PROGRAM MAIN
VAR
	pbGapMode: BOOL:=FALSE;
	pbTaperMode: BOOL:=FALSE;
	pbSingleCarrierMode: BOOL:=FALSE;
	pbDebugMode:BOOL:=FALSE;
	pbBCGapMode:BOOL:=FALSE;
	fb_led_Show: FB_LedShow;
	btn_reset: BOOL;
	CPMU_PLC_Reset: PLC_Reset;
	d_state: DINT;
	CPMU_PLC_Start: PLC_Start;
	powerStatus:BOOL;

(*TwinSAFE*)
	Safe_run AT%Q*:BOOL;
	Err_Ack AT %Q*:BOOL;
	Estop_RunAndRestart AT %Q*:BOOL;
	AX5805_Error_Ack AT %Q*:BOOL;
	Led_Run  AT %Q*:BOOL;
	Led_Error  AT %Q*:BOOL;

	FB_ERROR AT%I*:BOOL;
	COM_ERROR AT%I*:BOOL;
	//OUT_ERROR AT%I*:BOOL;
	Estop_Out AT%I*:BOOL;

	SafeStatus:INT;
	SafePLCRunOK: BOOL;
	fb_ton: TON;
	fb_ton2: TON;
	fb_ton3: TON;
	fb_ton1: TON;
	fb_ton0: TON;
(*IO*)
	el1808_D1  AT%I* :ARRAY[1..8] OF BOOL;
	el1008 AT%I*:BOOL;
	EStopTrig:BOOL;
(*setAxisPosition*)
	SetAxisPosState: INT;
	FB_Set_AxisPosition:FB_SetAxisPosition;
	fb_ton4: TON;
	fb_ton5: TON;
	fb_ton6: TON;
	SerAxisPositionDone: BOOL;

	i: INT;
	j: INT;

(****RS232***)
	fbEL6001	: FB_SerialCom;
	moveDoneLeftTop: BOOL;
	moveDoneRightTop: BOOL;
	moveDoneLeftBottom: BOOL;
	moveDoneRightBottom: BOOL;
	moveDoneAllAxis: BOOL;
	moveStatusLeftTop: BOOL;
	moveStatusRightTop: BOOL;
	moveStatusLeftBottom: BOOL;
	moveStatusRightBottom: BOOL;
	moveStatusAllAxis: BOOL;

(*Torque*)
	Torque_LT AT%I*:INT;
	Torque_RT AT%I*:INT;
	Torque_LB AT%I*:INT;
	Torque_RB AT%I*:INT;
(**)
	btn_setAxisPosition: BOOL;
	ValueSet_LeftTop:LREAL;
	ValueSet_RightTop:LREAL;
	ValueSet_LeftBottom:LREAL;
	ValueSet_RightBottom:LREAL;
(**)
	RestartTC: TC_Restart;
	
(*recipe*)
	RecipeINT:INT;
	RecipeBOOL:BOOL;
	RecipeManCommands: RecipeManCommands;
	SaveParameter : BOOL;  //保存文件
	LoadParameter : BOOL;  //读取文件
	Save_R_TRIG   : R_TRIG;
	Read_R_TRIG   : R_TRIG;
	loadparameterStatus: INT;
	RecipeBOOL2:BOOL;
	ReturnDwordLoad: DWORD;
	InsertionDeviceName:STRING;
(*UserMode*)
	pbUserMode: BOOL:=TRUE;
	EL1904 AT%I* :ARRAY[1..24] OF BOOL;
	setAxisPositionEnable: BOOL;
	state_loadParameters: INT;
	state_setLEPosBias: INT;
	//
	PositionBiasSet:BOOL;
	MC_SetLEPosBias_LeftTop:MC_WriteParameter;
	MC_SetLEPosBias_RightTop:MC_WriteParameter;
	MC_SetLEPosBias_LeftBottom:MC_WriteParameter;
	MC_SetLEPosBias_RightBottom:MC_WriteParameter;
	PositionBias_LeftTop: LREAL:=10.1;
	PositionBias_RightTop: LREAL:=10.2;
	PositionBias_LeftBottom: LREAL:=10.3;
	PositionBias_RightBottom: LREAL:=10.4;

	LoadLEPB_R_TRIG: R_TRIG;
	PositionBiasTON: TON;
	
	//
	OPC_TEST_Bi:BOOL:=TRUE; (*~ (OPC:1:available for OPC Clients) *)
	OPC_TEST_Bi2:BOOL;(*~ (OPC:1:available for OPC Clients) *)
	//
	HasTemperatureSensorOrNot:BOOL;//Only IVU or CPMU
	(*Sensor Reading*)
	Sensor_Reading_1 AT %I*:ARRAY[0..3] OF BYTE;
	Sensor_Reading_2 AT %I*:ARRAY[0..3] OF BYTE;
	Sensor_Reading_3 AT %I*:ARRAY[0..3] OF BYTE;
	Sensor_Reading_4 AT %I*:ARRAY[0..3] OF BYTE;
	Sensor_Reading_5 AT %I*:ARRAY[0..3] OF BYTE;
	Sensor_Reading_6 AT %I*:ARRAY[0..3] OF BYTE;
	Sensor_Reading_7 AT %I*:ARRAY[0..3] OF BYTE;
	Sensor_Reading_8 AT %I*:ARRAY[0..3] OF BYTE;
	Sensor_Reading_DpState AT %I*:USINT;
	Sensor_Reading_ExtDiagFlag AT %I*:BOOL;
	TemperatureSensors_1:LREAL;
	TemperatureSensors_2:LREAL;
	TemperatureSensors_3:LREAL;
	TemperatureSensors_4:LREAL;
	TemperatureSensors_5:LREAL;
	TemperatureSensors_6:LREAL;
	TemperatureSensors_7:LREAL;
	TemperatureSensors_8:LREAL;
	dut_sensor_datas_1:DUT_SENSOR_DATAS_1;
	dut_sensor_datas_2:DUT_SENSOR_DATAS_2;
	dut_sensor_datas_3:DUT_SENSOR_DATAS_3;
	dut_sensor_datas_4:DUT_SENSOR_DATAS_4;
	dut_sensor_datas_5:DUT_SENSOR_DATAS_5;
	dut_sensor_datas_6:DUT_SENSOR_DATAS_6;
	dut_sensor_datas_7:DUT_SENSOR_DATAS_7;
	dut_sensor_datas_8:DUT_SENSOR_DATAS_8;
	//
	temperature_gradient_2_To_1:LREAL;
	temperature_gradient_3_To_2:LREAL;
	temperature_gradient_5_To_4:LREAL;
	temperature_gradient_6_To_5:LREAL;
	temperature_gradient_max:LREAL;
	//
	temperature_average:LREAL;
	A_SetLinearEncoderPositionBias_Enable: BOOL;
	
		//
	temperatureStatus:INT;//0：有传感器度数错误；1:常温；2:低温；3:常温和低温中间态
	CryogenicTemperatureThreshold:LREAL:=80;//80K以下归划分为低温
	RoomTemperatureThreshold:LREAL:=293;//293K以上划分为常温
	//CPMU cryogenix ON/FF
	CryogenicCompensationOn:BOOL;
	CryogenicCompensationConditionsReady:BOOL;
	CryogenicCompensation_LeftTop:LREAL;
	CryogenicCompensation_RightTop:LREAL;
	CryogenicCompensation_LeftBottom:LREAL;
	CryogenicCompensation_RightBottom:LREAL;
	CryogenicCompensationDone: BOOL;
	
	(**)
	bDriveDiagMessageAndNumber  : BOOL;
	m_GetDriveStatusState:INT;
	GetDriveStatusStateDone:BOOL;
	GetDriveStatusStateError:BOOL;
	GetDriveStatusTON: TON;
	//	
	fb_SoEReadDiagMessage_LeftTop: FB_SoEReadDiagMessage;
	fb_SoEReadDiagMessage_RightTop: FB_SoEReadDiagMessage;
	fb_SoEReadDiagMessage_LeftBottom: FB_SoEReadDiagMessage;
	fb_SoEReadDiagMessage_RightBottom: FB_SoEReadDiagMessage;
	DriveDiagMessage_LeftTop:STRING;
	DriveDiagMessage_RightTop:STRING;
	DriveDiagMessage_LeftBottom:STRING;
	DriveDiagMessage_RightBottom:STRING;
	//
	FB_SoEReadDiagNumber_LeftTop: FB_SoEReadDiagNumber;
	FB_SoEReadDiagNumber_RightTop: FB_SoEReadDiagNumber;
	FB_SoEReadDiagNumber_LeftBottom: FB_SoEReadDiagNumber;
	FB_SoEReadDiagNumber_RightBottom: FB_SoEReadDiagNumber;
	DriveDiagNumber_LeftTop:UDINT;
	DriveDiagNumber_RightTop:UDINT;
	DriveDiagNumber_LeftBottom:UDINT;
	DriveDiagNumber_RightBottom:UDINT;
	bReloadDriveDiagMessageAndNumber: BOOL;
	
	(*load IOC*)
	bExe_load_Prog: BOOL;
	NT_StartProcess_Load: NT_StartProcess;
	Exe_load_step: UINT;
	R_TRIG_ExeLoad: R_TRIG;
	Exe_Load_Done:BOOL;
	(*kill IOC*)
	bExe_Kill_Prog: BOOL;
	NT_StartProcess_Kill: NT_StartProcess;
	Exe_kill_step: UINT;
	R_TRIG_Exekill: R_TRIG;
	Exe_Kill_Done:BOOL;
	LoadOpcIocTON:TON;
END_VAR

(*加载Ricipe参数*)
A_InitRecipeParameters();
(*Restart TwinCAT*)
IF Global_Variables.m_restartTC THEN
(*首先关闭opcIocShell.exe*)	
	bExe_Kill_Prog:=TRUE;
	A_KillOpcIocShellExe();
(*重启TC*)
	IF Exe_Kill_Done THEN
		A_RestartTC();
	END_IF
END_IF
(*******InitAxisParameters*******)
A_InitAxisParameters();
(*******CheckLimitSwitch*******)
A_CheckLimitSwitch();
(*Check Kill Switch*)
A_CheckKillSwitch();
(*******PosDiff¼à¿Ø*******)
A_PosDiffDetectiion();
(*******³õÊ¼»¯SafePlc*******)
IF NOT simulation THEN
A_SafePlcStartInit();
END_IF
(************SetAxisPosition*********************)
IF  NOT USELinearEncoder AND setAxisPositionEnable AND btn_setAxisPosition THEN
	//IF NOT SerAxisPositionDone THEN
		FB_Set_AxisPosition.ValueSet_LeftTop:=ValueSet_LeftTop;
		FB_Set_AxisPosition.ValueSet_RightTop:=ValueSet_RightTop;
		FB_Set_AxisPosition.ValueSet_LeftBottom:=ValueSet_LeftBottom;
		FB_Set_AxisPosition.ValueSet_RightBottom:=ValueSet_RightBottom;
		A_SetAxisPosition();
	//END_IF
END_IF
(*******³Mode Select******)
IF SafePLCRunOK OR Simulation THEN
	IF pbSingleCarrierMode AND NOT pbTaperMode AND NOT pbGapMode AND NOT pbDebugMode AND NOT pbBCGapMode AND NOT pbUserMode THEN
		SingleCarrierMode();
	ELSIF pbTaperMode  AND NOT pbSingleCarrierMode AND NOT pbGapMode  AND NOT pbDebugMode AND NOT pbBCGapMode AND NOT pbUserMode THEN
		TaperMode();
	ELSIF pbGapMode AND  NOT pbSingleCarrierMode AND NOT pbTaperMode  AND NOT pbDebugMode AND NOT pbBCGapMode AND NOT pbUserMode THEN
		GapMode();
	ELSIF pbDebugMode AND NOT pbGapMode AND NOT pbSingleCarrierMode AND NOT pbTaperMode AND NOT pbBCGapMode  AND NOT pbUserMode THEN
		DebugMode();
	ELSIF pbBCGapMode AND NOT pbGapMode AND NOT pbSingleCarrierMode AND NOT pbTaperMode AND NOT pbDebugMode AND NOT pbUserMode THEN
		BCGapMode();
	ELSIF pbUserMode AND NOT pbGapMode AND NOT pbSingleCarrierMode AND NOT pbTaperMode AND NOT pbDebugMode AND NOT pbBCGapMode THEN
		UserMode();
	END_IF
END_IF
(*******Led Show******)
fb_led_Show();
(*******Check Power status******)
FB_Power(Check:=TRUE);
st_Power:=FB_Power.PowerState;
(******Check Couple Status*****)
FB_CheckCoupleStatus(Check:=TRUE);
st_Couple:=FB_CheckCoupleStatus.CoupleState;
(*********RS232*********************)
BackgroundEL();
(*fbEL6001(TxBuffer:=TxBufferEL, RxBuffer:=RxBufferEL);*)

(*获取温度传感器数据*)
A_GetTemperatureSensorsData();
(*低温补偿监控*)
A_CryogenicCompensationMonitoring();

(*设置position bias*)
IF loadParametersDone AND (DriveStatus=1 OR simulation) THEN 
	A_SetLinearEncoderPositionBias();
END_IF
(*检查硬急停状态，包括安全限位、柜门急停、手持急停*)
A_CheckHardwareEmergencyStopStatus();
(*获取驱动器状态信息*)
IF NOT simulation THEN
	A_GetDriverStatus();
END_IF
(*IDControlReady*)
IF ((DriveStatus<>0 AND SafePLCRunOK) OR simulation) AND NOT Error THEN
//IF (SafePLCRunOK OR simulation) AND NOT Error THEN
	IDControlReady:=TRUE;
ELSE
	IDControlReady:=FALSE;
END_IF

(*IOC Start*)
IF SafePLCRunOK OR simulation THEN
	bExe_load_Prog:=TRUE;
	A_LoadOpcIocShellExe();
END_IF

ACTION A_CheckHardwareEmergencyStopStatus:
IF 	NOT KS_LeftTop_Far_Contact1 OR
	NOT KS_LeftTop_Far_Contact2 OR
	NOT KS_RightTop_Far_Contact1 OR
	NOT KS_RightTop_Far_Contact2 OR
	NOT KS_LeftBottom_Far_Contact1 OR
	NOT KS_LeftBottom_Far_Contact2 OR
	NOT KS_RightBottom_Far_Contact1 OR
	NOT KS_RightBottom_Far_Contact2 OR
	
	NOT KS_LeftTop_Near_Contact1 OR
	NOT KS_LeftTop_Near_Contact2 OR
	NOT KS_RightTop_Near_Contact1 OR
	NOT KS_RightTop_Near_Contact2 OR
	NOT KS_LeftBottom_Near_Contact1 OR
	NOT KS_LeftBottom_Near_Contact2 OR
	NOT KS_RightBottom_Near_Contact1 OR
	NOT KS_RightBottom_Near_Contact2 OR
(*E-STOP*)
	NOT KS_CabinetEmergency_contact1 OR
	NOT KS_CabinetEmergency_contact2 OR
	NOT KS_handEmergency1_Contact1 OR
	NOT KS_handEmergency1_Contact2 OR
	NOT KS_handEmergency2_Contact1 OR
	NOT KS_handEmergency2_Contact2 OR
	NOT KS_softEmergency2_Contact THEN
	Hardware_EmergencyStop:=FALSE;
ELSE
	Hardware_EmergencyStop:=TRUE;
END_IF
END_ACTION

ACTION A_CheckKillSwitch:
IF simulation THEN
	KS_LeftTop_Far_Contact1:=TRUE;
	KS_LeftTop_Far_Contact2:=TRUE;
	KS_LeftTop_Near_Contact1:=TRUE;
	KS_LeftTop_Near_Contact2:=TRUE;
	KS_RightTop_Far_Contact1:=TRUE;
	KS_RightTop_Far_Contact2:=TRUE;
	KS_RightTop_Near_Contact1:=TRUE;
	KS_RightTop_Near_Contact2:=TRUE;
	KS_LeftBottom_Far_Contact1:=TRUE;
	KS_LeftBottom_Far_Contact2:=TRUE;
	KS_LeftBottom_Near_Contact1:=TRUE;
	KS_LeftBottom_Near_Contact2:=TRUE;	
	KS_RightBottom_Far_Contact1:=TRUE;
	KS_RightBottom_Far_Contact2:=TRUE;
	KS_RightBottom_Near_Contact1:=TRUE;
	KS_RightBottom_Near_Contact2:=TRUE;		
	(*E-STOP*)
	KS_CabinetEmergency_contact1:=TRUE;
	KS_CabinetEmergency_contact2:=TRUE;	
	KS_handEmergency1_Contact1:=TRUE;
	KS_handEmergency1_Contact2:=TRUE;
	KS_handEmergency2_Contact1:=TRUE;
	KS_handEmergency2_Contact2:=TRUE;
	
	KS_softEmergency2_Contact:=TRUE;

ELSE
	KS_LeftTop_Far_Contact1:=EL1904[1];//c1
	KS_LeftTop_Far_Contact2:=EL1904[2];//c2
	KS_LeftTop_Near_Contact1:=EL1904[3];//c3
	KS_LeftTop_Near_Contact2:=EL1904[4];//c4
	
	KS_RightTop_Far_Contact1:=EL1904[5];
	KS_RightTop_Far_Contact2:=EL1904[6];
	KS_RightTop_Near_Contact1:=EL1904[7];
	KS_RightTop_Near_Contact2:=EL1904[8];
	
	KS_LeftBottom_Far_Contact1:=EL1904[9];
	KS_LeftBottom_Far_Contact2:=EL1904[10];
	KS_LeftBottom_Near_Contact1:=EL1904[11];
	KS_LeftBottom_Near_Contact2:=EL1904[12];
	
	KS_RightBottom_Far_Contact1:=EL1904[13];
	KS_RightBottom_Far_Contact2:=EL1904[14];
	KS_RightBottom_Near_Contact1:=EL1904[15];
	KS_RightBottom_Near_Contact2:=EL1904[16];	
	
	
	(*E-STOP*)
	KS_CabinetEmergency_contact1:=EL1904[17];
	KS_CabinetEmergency_contact2:=EL1904[18];
	
	KS_handEmergency1_Contact1:=EL1904[19];
	KS_handEmergency1_Contact2:=EL1904[20];
	KS_handEmergency2_Contact1:=EL1904[21];
	KS_handEmergency2_Contact2:=EL1904[22];
	
	KS_softEmergency2_Contact:=EL1904[23];
	END_IF
END_ACTION

ACTION A_CheckLimitSwitch:
(*******1.´ÓIO»ñÈ¡ÏÞÎ»×´Ì¬******)
(**)
IF simulation THEN
	(**)
	LS_LeftTop_Top:=TRUE;
	LS_LeftTop_Bottom:=TRUE;
	LS_RightTop_Top:=TRUE;
	LS_RightTop_Bottom:=TRUE;
	LS_LeftBottom_Top:=TRUE;
	LS_LeftBottom_Bottom:=TRUE;
	LS_RightBottom_Top:=TRUE;
	LS_RightBottom_Bottom:=TRUE;
ELSE
	LS_LeftTop_Top :=el1808_D1[1];
	LS_LeftTop_Bottom:=el1808_D1[3];
	LS_RightTop_Top:=el1808_D1[2];
	LS_RightTop_Bottom:=el1808_D1[4];
	LS_LeftBottom_Top:=el1808_D1[7];
	LS_LeftBottom_Bottom:=el1808_D1[5];
	LS_RightBottom_Top:=el1808_D1[8];
	LS_RightBottom_Bottom:=el1808_D1[6];
END_IF
(*
	LS_LeftTop_Top:=TRUE;
	LS_LeftTop_Bottom:=TRUE;
	LS_RightTop_Top:=TRUE;
	LS_RightTop_Bottom:=TRUE;
	LS_LeftBottom_Top:=TRUE;
	LS_LeftBottom_Bottom:=TRUE;
	LS_RightBottom_Top:=TRUE;
	LS_RightBottom_Bottom:=TRUE;
*)
(******2.TopÏÞÎ»»òÕßBottomÏÞÎ»ÓÐÒ»¸ö´¥·¢£¬È«¾Ö±äÁ¿¡£¸øMC_POWERÓÃÓÚ·½Ïò¿ØÖÆ£¬ÓÐÒ»¸öÏÞÎ»Îª´¥·¢ÎªFALSE£¬ÔòUnreach_LSÎªFALSE******)
Unreach_LS_Top:=LS_LeftTop_Top AND LS_RightTop_Top AND LS_LeftBottom_Top AND LS_RightBottom_Top;
Unreach_LS_Bottom:=LS_LeftTop_Bottom AND LS_RightTop_Bottom AND LS_LeftBottom_Bottom AND LS_RightBottom_Bottom;
(**************************ÏòTopÔË¶¯Ê±£¬´¥ÅöBottomÏÞÎ»¿ª¹Ø£¬»òÕßÏà·´£¬ESTOP**************************************)
(*
IF LeftTopLin.Status.Moving AND Velo_LeftTopLin>0 THEN
	IF NOT Unreach_LS_Bottom THEN
		Error:=TRUE;
		ErrorID:=61;
		FB_PlcEmergencyStop();
	END_IF
ELSIF LeftTopLin.Status.Moving AND Velo_LeftTopLin<0 THEN
	IF NOT Unreach_LS_Top THEN
		Error:=TRUE;
		ErrorID:=62;
		FB_PlcEmergencyStop();
	END_IF
ELSIF RightTopLin.Status.Moving AND Velo_RightTopLin>0 THEN
	IF NOT Unreach_LS_Bottom THEN
		Error:=TRUE;
		ErrorID:=63;
		FB_PlcEmergencyStop();
	END_IF
ELSIF RightTopLin.Status.Moving AND Velo_RightTopLin<0 THEN
	IF NOT  Unreach_LS_Top THEN
		Error:=TRUE;
		ErrorID:=64;
		FB_PlcEmergencyStop();
	END_IF
ELSIF LeftBottomLin.Status.Moving AND Velo_LeftBottomLin>0 THEN
	IF NOT Unreach_LS_Bottom THEN
		Error:=TRUE;
		ErrorID:=65;
		FB_PlcEmergencyStop();
	END_IF
ELSIF LeftBottomLin.Status.Moving AND Velo_LeftBottomLin<0 THEN
	IF NOT Unreach_LS_Top THEN
		Error:=TRUE;
		ErrorID:=66;
		FB_PlcEmergencyStop();
	END_IF
ELSIF RightBottomLin.Status.Moving AND Velo_RightBottomLin>0 THEN
	IF NOT Unreach_LS_Bottom THEN
		Error:=TRUE;
		ErrorID:=67;
		FB_PlcEmergencyStop();
	END_IF
ELSIF RightBottomLin.Status.Moving AND Velo_RightBottomLin<0 THEN
	IF NOT Unreach_LS_Top THEN
		Error:=TRUE;
		ErrorID:=68;
		FB_PlcEmergencyStop();
	END_IF
END_IF
*)
(*
(******3.ÓÐÒ»¸öÏÞÎ»´¥·¢£¬ delayÊ±¼äºó£¬¼à²âÖáÊÇ·ñÔÚÍ£Ö¹×´Ì¬£¬ÈôÃ»ÓÐ£¬Emergency AND PowerOff******)
IF NOT Unreach_LS_Top OR NOT Unreach_LS_Bottom THEN
	fb_ton.IN:=TRUE;
END_IF
IF fb_ton.Q THEN
	IF LeftTopLin.Status.Moving OR RightTopLin.Status.Moving OR LeftBottomLin.Status.Moving OR RightBottomLin.Status.Moving THEN
		FB_PlcEmergencyStop();
		fb_ton.IN:=FALSE;
		Error:=TRUE;
		EStopTrig:=TRUE;
		ErrorID:=1;
		(*FB_Power_Off(Execute:=TRUE);*)
	END_IF
END_IF

(*******4.µ¥ÖáÉÏÏÂÏÞÎ»¾ùÎªFALSEÊ±£¬ÏÞÎ»´íÎó£¬Emergency*******)
IF (NOT LS_LeftTop_Top AND NOT LS_LeftTop_Bottom) OR  (NOT  LS_RightTop_Top AND NOT LS_RightTop_Bottom)
		OR (NOT LS_LeftBottom_Top AND NOT LS_LeftBottom_Bottom) OR (NOT LS_RightBottom_Top AND NOT LS_RightBottom_Bottom) THEN
	(*FB_Plc_EmergencyStop();*)
	Error:=TRUE;
	EStopTrig:=TRUE;
	ErrorID:=2;
END_IF
*)
END_ACTION

ACTION A_CryogenicCompensationMonitoring:
//没有传感器OR不是CPMU不低温补偿OR低温不到位，均不补偿
IF NOT HasTemperatureSensorOrNot OR NOT CryogenicCompensationOn THEN //OR temperatureStatus<>2 THEN
	//不补偿
	CryogenicCompensation_LeftTop:=0;
	CryogenicCompensation_RightTop:=0;
	CryogenicCompensation_LeftBottom:=0;
	CryogenicCompensation_RightBottom:=0;
ELSE
	CryogenicCompensationConditionsReady:=TRUE;//条件具备，可以低温补偿
	//检查补偿值，单轴补偿范围均在0-1内
	IF CryogenicCompensation_LeftTop>1 OR CryogenicCompensation_LeftTop<=0 THEN
			Error:=TRUE;
			ErrorID:=1201;
			ErrorDescription:='CryogenicCompensation_LeftTop>1 OR CryogenicCompensation_LeftTop<=0';
			FB_PlcEmergencyStop();
	END_IF
	IF CryogenicCompensation_RightTop>1 OR CryogenicCompensation_RightTop<=0 THEN
			Error:=TRUE;
			ErrorID:=1202;
			ErrorDescription:='CryogenicCompensation_RightTop>1 OR CryogenicCompensation_RightTop<=0';
			FB_PlcEmergencyStop();
	END_IF
	IF CryogenicCompensation_LeftBottom>1 OR CryogenicCompensation_LeftBottom<=0 THEN
			Error:=TRUE;
			ErrorID:=1203;
			ErrorDescription:='CryogenicCompensation_LeftBottom>1 OR CryogenicCompensation_LeftBottom<=0';
			FB_PlcEmergencyStop();
	END_IF
	IF CryogenicCompensation_RightBottom>1 OR CryogenicCompensation_RightBottom<=0 THEN
			Error:=TRUE;
			ErrorID:=1204;
			ErrorDescription:='CryogenicCompensation_RightBottom>1 OR CryogenicCompensation_RightBottom<=0';
			FB_PlcEmergencyStop();
	END_IF
END_IF
//若在低温补偿模式，但是温度没到低温区间，则Emergency，不允许启动
(*
IF CryogenicCompensationOn AND temperatureStatus<>2 THEN
			Error:=TRUE;
			ErrorID:=1205;
			ErrorDescription:='CryogenicCompensationOn AND temperatureStatus<>2';
			FB_PlcEmergencyStop();
END_IF
*)
END_ACTION

ACTION A_GetDriverStatus:
IF bReloadDriveDiagMessageAndNumber THEN
	m_GetDriveStatusState:=0;
	bReloadDriveDiagMessageAndNumber:=FALSE;
END_IF
GetDriveStatusTON(PT:=T#1S);
A_GetDriverStatusMC();
CASE m_GetDriveStatusState OF
	0:
		GetDriveStatusTON.IN:=TRUE;
		m_GetDriveStatusState:=1;
	1:
		IF GetDriveStatusTON.Q THEN
			bDriveDiagMessageAndNumber:=TRUE;
			m_GetDriveStatusState:=2;
		END_IF
	2:
		GetDriveStatusTON.IN:=FALSE;
		DriveDiagMessage_LeftTop:=fb_SoEReadDiagMessage_LeftTop.sDiagMessage.strData;
		DriveDiagMessage_RightTop:=fb_SoEReadDiagMessage_RightTop.sDiagMessage.strData;
		DriveDiagMessage_LeftBottom:=fb_SoEReadDiagMessage_LeftBottom.sDiagMessage.strData;
		DriveDiagMessage_RightBottom:=fb_SoEReadDiagMessage_RightBottom.sDiagMessage.strData;
		//
		DriveDiagNumber_LeftTop:=FB_SoEReadDiagNumber_LeftTop.iDiagNumber;
		DriveDiagNumber_RightTop:=FB_SoEReadDiagNumber_RightTop.iDiagNumber;
		DriveDiagNumber_LeftBottom:=FB_SoEReadDiagNumber_LeftBottom.iDiagNumber;
		DriveDiagNumber_RightBottom:=FB_SoEReadDiagNumber_RightBottom.iDiagNumber;
		//
		IF 	NOT fb_SoEReadDiagMessage_LeftTop.bBusy
			AND NOT fb_SoEReadDiagMessage_RightTop.bBusy
			AND NOT fb_SoEReadDiagMessage_LeftBottom.bBusy
			AND NOT fb_SoEReadDiagMessage_RightBottom.bBusy 
			AND NOT FB_SoEReadDiagNumber_LeftTop.bBusy
			AND NOT  FB_SoEReadDiagNumber_RightTop.bBusy
			AND NOT FB_SoEReadDiagNumber_LeftBottom.bBusy
			AND NOT FB_SoEReadDiagNumber_RightBottom.bBusy THEN
			m_GetDriveStatusState:=88;
		END_IF
		IF 	fb_SoEReadDiagMessage_LeftTop.bError
			OR fb_SoEReadDiagMessage_RightTop.bError
			OR fb_SoEReadDiagMessage_LeftBottom.bError
			OR fb_SoEReadDiagMessage_RightBottom.bError
			OR FB_SoEReadDiagNumber_LeftTop.bError
			OR FB_SoEReadDiagNumber_RightTop.bError
			OR FB_SoEReadDiagNumber_LeftBottom.bError
			OR FB_SoEReadDiagNumber_RightBottom.bError THEN
			m_GetDriveStatusState:=-100;
		END_IF
		(*Drive Status*)
		//D012, Axis state machine: Control and power section ready
		IF DriveDiagNumber_LeftTop=16#D012 AND DriveDiagNumber_RightTop=16#D012
			AND DriveDiagNumber_LeftBottom=16#D012 AND DriveDiagNumber_RightBottom=16#D012 THEN
			DriveStatus:=1;
		//D013, Axis state machine: Axis in operation
		ELSIF DriveDiagNumber_LeftTop=16#D013 AND DriveDiagNumber_RightTop=16#D013
			AND DriveDiagNumber_LeftBottom=16#D013 AND DriveDiagNumber_RightBottom=16#D013 THEN
			DriveStatus:=2;
		ELSE
			DriveStatus:=0;
		END_IF
	88:
		bDriveDiagMessageAndNumber:=FALSE;
		A_GetDriverStatusMC();
		GetDriveStatusStateDone:=TRUE;
		GetDriveStatusStateError:=FALSE;
		m_GetDriveStatusState:=0;
	-100:
		bDriveDiagMessageAndNumber:=FALSE;
		A_GetDriverStatusMC();
		GetDriveStatusStateDone:=FALSE;
		GetDriveStatusStateError:=TRUE;
		Error:=TRUE;
		ErrorId:=1301;
		ErrorDescription:='GetDriveStatusStateError';
END_CASE


(*IF bDriveDiagNumber THEN
    fbDriveDiagNumber_LeftTop(
       Axis     := LeftTopLin.NcToPlc,
       bExecute := TRUE,
       tTimeout := DEFAULT_ADS_TIMEOUT,
       iDiagNumber =>DriveDiagNumber_LeftTop
    );
    IF NOT fbDriveDiagNumber_LeftTop.bBusy THEN
        fbDriveDiagNumber_LeftTop(Axis := LeftTopLin.NcToPlc, bExecute := FALSE);
        bDriveDiagNumber := FALSE;
    END_IF
END_IF

IF bDriveDiagMessage THEN
    fbDriveDiagMessage_LeftTop(
       Axis     := LeftTopLin.NcToPlc,
       bExecute := TRUE,
       tTimeout := DEFAULT_ADS_TIMEOUT,
       sDiagMessage=>DriveDiagMessage_LeftTop
    );
    IF NOT fbDriveDiagMessage_LeftTop.bBusy THEN
        fbDriveDiagMessage_LeftTop(Axis := LeftTopLin.NcToPlc, bExecute := FALSE);
        bDriveDiagMessage := FALSE;
    END_IF
	DriveDiagMessageString_LeftTop:=DriveDiagMessage_LeftTop.strData;
END_IF
*)
END_ACTION

ACTION A_GetDriverStatusMC:
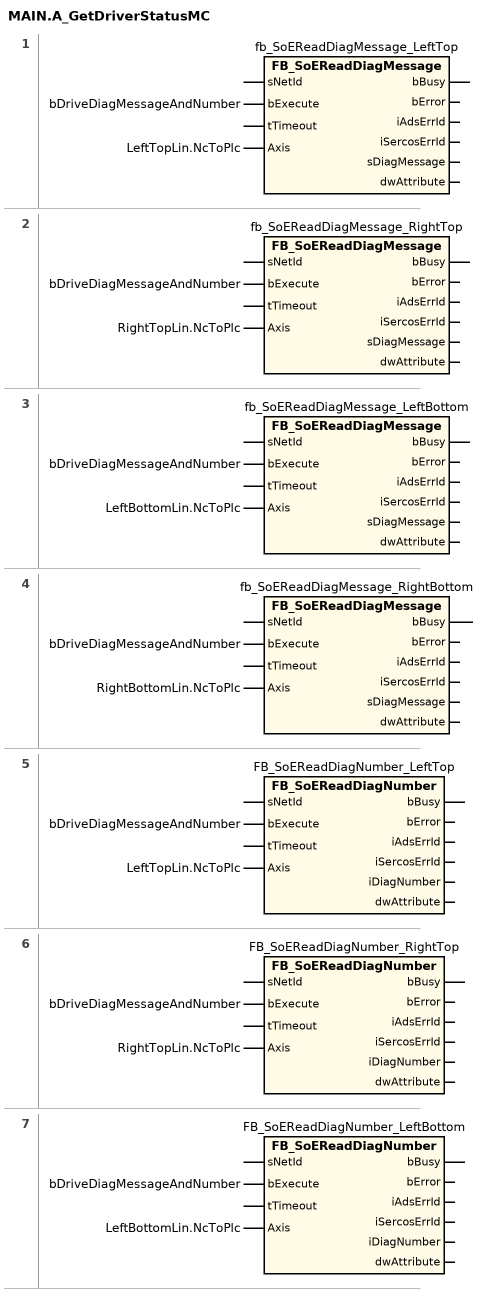
// NETWORK 1
fb_SoEReadDiagMessage_LeftTop(bExecute := bDriveDiagMessageAndNumber, Axis := LeftTopLin.NcToPlc); // FB_SoEReadDiagMessage

// NETWORK 2
fb_SoEReadDiagMessage_RightTop(bExecute := bDriveDiagMessageAndNumber, Axis := RightTopLin.NcToPlc); // FB_SoEReadDiagMessage

// NETWORK 3
fb_SoEReadDiagMessage_LeftBottom(bExecute := bDriveDiagMessageAndNumber, Axis := LeftBottomLin.NcToPlc); // FB_SoEReadDiagMessage

// NETWORK 4
fb_SoEReadDiagMessage_RightBottom(bExecute := bDriveDiagMessageAndNumber, Axis := RightBottomLin.NcToPlc); // FB_SoEReadDiagMessage

// NETWORK 5
FB_SoEReadDiagNumber_LeftTop(bExecute := bDriveDiagMessageAndNumber, Axis := LeftTopLin.NcToPlc); // FB_SoEReadDiagNumber

// NETWORK 6
FB_SoEReadDiagNumber_RightTop(bExecute := bDriveDiagMessageAndNumber, Axis := RightTopLin.NcToPlc); // FB_SoEReadDiagNumber

// NETWORK 7
FB_SoEReadDiagNumber_LeftBottom(bExecute := bDriveDiagMessageAndNumber, Axis := LeftBottomLin.NcToPlc); // FB_SoEReadDiagNumber

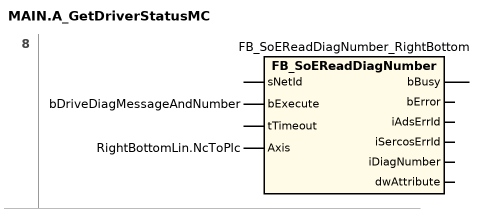
// NETWORK 8
FB_SoEReadDiagNumber_RightBottom(bExecute := bDriveDiagMessageAndNumber, Axis := RightBottomLin.NcToPlc); // FB_SoEReadDiagNumber
END_ACTION

ACTION A_GetTemperatureSensorsData:
//sensor_1
dut_sensor_datas_1.data_byte[3]:=Sensor_Reading_1[0];
dut_sensor_datas_1.data_byte[2]:=Sensor_Reading_1[1];
dut_sensor_datas_1.data_byte[1]:=Sensor_Reading_1[2];
dut_sensor_datas_1.data_byte[0]:=Sensor_Reading_1[3];
TemperatureSensors_1:=DINT_TO_LREAL(LREAL_TO_DINT(dut_sensor_datas_1.data_lreal*100))/100;
//sensor_2
dut_sensor_datas_2.data_byte[3]:=Sensor_Reading_2[0];
dut_sensor_datas_2.data_byte[2]:=Sensor_Reading_2[1];
dut_sensor_datas_2.data_byte[1]:=Sensor_Reading_2[2];
dut_sensor_datas_2.data_byte[0]:=Sensor_Reading_2[3];
TemperatureSensors_2:=DINT_TO_LREAL(LREAL_TO_DINT(dut_sensor_datas_2.data_lreal*100))/100;
//sensor_3
dut_sensor_datas_3.data_byte[3]:=Sensor_Reading_3[0];
dut_sensor_datas_3.data_byte[2]:=Sensor_Reading_3[1];
dut_sensor_datas_3.data_byte[1]:=Sensor_Reading_3[2];
dut_sensor_datas_3.data_byte[0]:=Sensor_Reading_3[3];
TemperatureSensors_3:=DINT_TO_LREAL(LREAL_TO_DINT(dut_sensor_datas_3.data_lreal*100))/100;
//sensor_4
dut_sensor_datas_4.data_byte[3]:=Sensor_Reading_4[0];
dut_sensor_datas_4.data_byte[2]:=Sensor_Reading_4[1];
dut_sensor_datas_4.data_byte[1]:=Sensor_Reading_4[2];
dut_sensor_datas_4.data_byte[0]:=Sensor_Reading_4[3];
TemperatureSensors_4:=DINT_TO_LREAL(LREAL_TO_DINT(dut_sensor_datas_4.data_lreal*100))/100;
//sensor_5
dut_sensor_datas_5.data_byte[3]:=Sensor_Reading_5[0];
dut_sensor_datas_5.data_byte[2]:=Sensor_Reading_5[1];
dut_sensor_datas_5.data_byte[1]:=Sensor_Reading_5[2];
dut_sensor_datas_5.data_byte[0]:=Sensor_Reading_5[3];
TemperatureSensors_5:=DINT_TO_LREAL(LREAL_TO_DINT(dut_sensor_datas_5.data_lreal*100))/100;
//sensor_6
dut_sensor_datas_6.data_byte[3]:=Sensor_Reading_6[0];
dut_sensor_datas_6.data_byte[2]:=Sensor_Reading_6[1];
dut_sensor_datas_6.data_byte[1]:=Sensor_Reading_6[2];
dut_sensor_datas_6.data_byte[0]:=Sensor_Reading_6[3];
TemperatureSensors_6:=DINT_TO_LREAL(LREAL_TO_DINT(dut_sensor_datas_6.data_lreal*100))/100;
//sensor_7
dut_sensor_datas_7.data_byte[3]:=Sensor_Reading_7[0];
dut_sensor_datas_7.data_byte[2]:=Sensor_Reading_7[1];
dut_sensor_datas_7.data_byte[1]:=Sensor_Reading_7[2];
dut_sensor_datas_7.data_byte[0]:=Sensor_Reading_7[3];
TemperatureSensors_7:=DINT_TO_LREAL(LREAL_TO_DINT(dut_sensor_datas_7.data_lreal*100))/100;
//sensor_8
dut_sensor_datas_8.data_byte[3]:=Sensor_Reading_8[0];
dut_sensor_datas_8.data_byte[2]:=Sensor_Reading_8[1];
dut_sensor_datas_8.data_byte[1]:=Sensor_Reading_8[2];
dut_sensor_datas_8.data_byte[0]:=Sensor_Reading_8[3];
TemperatureSensors_8:=DINT_TO_LREAL(LREAL_TO_DINT(dut_sensor_datas_8.data_lreal*100))/100;
//计算temperature_gradient
temperature_gradient_2_To_1:=ABS(TemperatureSensors_2-TemperatureSensors_1);
temperature_gradient_3_To_2:=ABS(TemperatureSensors_3-TemperatureSensors_2);
temperature_gradient_5_To_4:=ABS(TemperatureSensors_5-TemperatureSensors_4);
temperature_gradient_6_To_5:=ABS(TemperatureSensors_6-TemperatureSensors_5);
temperature_gradient_max:=DINT_TO_LREAL(LREAL_TO_DINT(MAX(temperature_gradient_2_To_1,temperature_gradient_3_To_2,
							temperature_gradient_5_To_4,temperature_gradient_6_To_5)*100))/100;
//计算大梁上的温度平均值
temperature_average:=DINT_TO_LREAL(LREAL_TO_DINT((TemperatureSensors_1+TemperatureSensors_2+TemperatureSensors_3+TemperatureSensors_4
					+TemperatureSensors_5+TemperatureSensors_6)/6*100))/100;
					

//传感器温度状态：0：有传感器度数错误；1:常温；2:低温；3:常温和低温中间态
IF TemperatureSensors_1=0 OR TemperatureSensors_2=0 OR TemperatureSensors_3=0 
	OR TemperatureSensors_4=0 OR TemperatureSensors_5=0 OR TemperatureSensors_6=0 THEN	
	temperatureStatus:=0;//有传感器读数错误
ELSIF TemperatureSensors_1>=RoomTemperatureThreshold AND TemperatureSensors_2>=RoomTemperatureThreshold AND TemperatureSensors_3>=RoomTemperatureThreshold
	AND TemperatureSensors_4>=RoomTemperatureThreshold AND TemperatureSensors_5>=RoomTemperatureThreshold AND TemperatureSensors_6>=RoomTemperatureThreshold THEN	
	temperatureStatus:=1;//常温
ELSIF TemperatureSensors_1<=CryogenicTemperatureThreshold AND TemperatureSensors_1>77
	AND TemperatureSensors_2<=CryogenicTemperatureThreshold  AND TemperatureSensors_2>77
	AND TemperatureSensors_3<=CryogenicTemperatureThreshold  AND TemperatureSensors_3>77
	AND TemperatureSensors_4<=CryogenicTemperatureThreshold   AND TemperatureSensors_4>77
	AND TemperatureSensors_5<=CryogenicTemperatureThreshold  AND TemperatureSensors_5>77
	AND TemperatureSensors_6<=CryogenicTemperatureThreshold   AND TemperatureSensors_6>77 THEN	
	temperatureStatus:=2;//低温
ELSE
	temperatureStatus:=3;//常温和低温中间
END_IF
END_ACTION

ACTION A_InitAxisParameters:
(*ÖáÎ»ÖÃ¡¢ËÙ¶È¡¢PosDiff*)

	Pos_LeftTopLin:=DINT_TO_LREAL(LREAL_TO_DINT(LeftTopLin.NcToPlc.ActPos*100000))/100000;
	Pos_RightTopLin:=DINT_TO_LREAL(LREAL_TO_DINT(RightTopLin.NcToPlc.ActPos*100000))/100000;
	Pos_LeftBottomLin:=DINT_TO_LREAL(LREAL_TO_DINT(LeftBottomLin.NcToPlc.ActPos*100000))/100000;
	Pos_RightBottomLin:=DINT_TO_LREAL(LREAL_TO_DINT(RightBottomLin.NcToPlc.ActPos*100000))/100000;

	
	LB_TestRecord:=Pos_LeftBottomLin-5;
	RB_TestRecord:=Pos_RightBottomLin-5;
	moveStatusLeftTop:=LeftTopLin.Status.Moving;
	moveStatusRightTop:=RightTopLin.Status.Moving;
	moveStatusLeftBottom:=LeftBottomLin.Status.Moving;
	moveStatusRightBottom:=RightBottomLin.Status.Moving;
	moveStatusAllAxis:=moveStatusLeftTop AND moveStatusRightTop AND moveStatusLeftBottom AND moveStatusRightBottom;

	Velo_LeftTopLin:=DINT_TO_LREAL(LREAL_TO_DINT(LeftTopLin.NcToPlc.ActVelo*100000))/100000;
	Velo_RightTopLin:=DINT_TO_LREAL(LREAL_TO_DINT(RightTopLin.NcToPlc.ActVelo*100000))/100000;
	Velo_LeftBottomLin:=DINT_TO_LREAL(LREAL_TO_DINT(LeftBottomLin.NcToPlc.ActVelo*100000))/100000;
	Velo_RightBottomLin:=DINT_TO_LREAL(LREAL_TO_DINT(RightBottomLin.NcToPlc.ActVelo*100000))/100000;

	PosDiff_LeftTopLin_actual:=LeftTopLin.NcToPlc.PosDiff;
	PosDiff_RightTopLin_actual:=RightTopLin.NcToPlc.PosDiff;
	PosDiff_LeftBottomLin_actual:=LeftBottomLin.NcToPlc.PosDiff;
	PosDiff_RightBottomLin_actual:=RightBottomLin.NcToPlc.PosDiff;

	LeftTopLin.ReadStatus();
	RightTopLin.ReadStatus();
	LeftBottomLin.ReadStatus();
	RightBottomLin.ReadStatus();
END_ACTION

ACTION A_InitRecipeParameters:
CASE state_loadParameters OF
	0:
		LoadParameter:=TRUE;
		Read_R_TRIG(CLK:=LoadParameter , Q=> );
		IF Read_R_TRIG.Q THEN
			state_loadParameters:=1;
		END_IF
	1:
		 ReturnDwordLoad:=RecipeManCommands.LoadAndWriteRecipe(RecipeDefinitionName:='Recipes' , RecipeName:='Parameters');
    	 LoadParameter:=FALSE;
		 IF ReturnDwordLoad<>0 THEN
		 	state_loadParameters:=-100;
		ELSE
			LoadRecipeParameters:=TRUE;
			LoadParameter:=FALSE;
			state_loadParameters:=88;
	 	END_IF
	88:
		loadParametersDone:=TRUE;
	-100:
		loadParametersDone:=FALSE;
		Error:=TRUE;
		ErrorId:=101;
		ErrorDescription:='LoadRecipeParameters Error';
		Plc_EmergencyStop:=FALSE;
END_CASE

////Save_R_TRIG(CLK:=SaveParameter , Q=> );
//Read_R_TRIG(CLK:=LoadParameter , Q=> );
//IF Save_R_TRIG.Q THEN  //将plc数据以文件形式保存在工控机中
//	 RecipeManCommands.CreateRecipe(RecipeDefinitionName:='Recipes' , RecipeName:='Parameters' );
//	 RecipeManCommands.ReadAndSaveRecipe(RecipeDefinitionName:='Recipes' , RecipeName:='Parameters' );
//	 SaveParameter:=FALSE;
//END_IF
//IF Read_R_TRIG.Q THEN  //将工控机中的文件数据读取到plc中
//     ReturnDwordLoad:=RecipeManCommands.LoadAndWriteRecipe(RecipeDefinitionName:='Recipes' , RecipeName:='Parameters');
//     LoadParameter:=FALSE;
//	 IF ReturnDwordLoad<>0 THEN
//		 Error:=TRUE;
//		 ErrorId:=101;
//		 ErrorDescription:='LoadRecipeParameters Error';
//		 Plc_EmergencyStop:=FALSE;
//	 END_IF
//END_IF
END_ACTION

ACTION A_KillOpcIocShellExe:
R_TRIG_Exekill(CLK:=bExe_Kill_Prog, Q=> );
CASE Exe_kill_step OF
	0:
		IF R_TRIG_Exekill.Q THEN
			NT_StartProcess_Kill.START:=FALSE;
			NT_StartProcess_Kill.PATHSTR:='C:\HZB\OpcIocShell\IDControlIOC\killcmd.bat';
			//NT_StartProcess_Kill.DIRNAME:='C:\Program Files (x86)\HZB\OpcIocShell\bin\opcIocShell.exe';
			Exe_kill_step:=10;
		END_IF;
	10:
		NT_StartProcess_Kill.START:=TRUE;
		Exe_kill_step:=20;
	20:
		IF NT_StartProcess_Kill.ERR THEN
			Exe_kill_step:=0;
		ELSE
			Exe_kill_step:=30;
		END_IF;

	30:
		NT_StartProcess_Kill.START:=TRUE;
		Exe_kill_step:=40;
	40:
		IF NOT NT_StartProcess_Kill.BUSY THEN
			NT_StartProcess_Kill.START:=FALSE;
			Exe_Kill_Done:=TRUE;
			Exe_kill_step:=0;
		END_IF;
END_CASE;

NT_StartProcess_Kill(
	NETID:='' ,
	PATHSTR:= ,
	DIRNAME:= , 
	COMNDLINE:= , 
	START:= ,
	ERRID=> );
END_ACTION

ACTION A_LoadOpcIocShellExe:
R_TRIG_Exeload(CLK:=bExe_load_Prog, Q=> );
LoadOpcIocTON(PT:=T#10S);
CASE Exe_load_step OF
	0:
		LoadOpcIocTON.IN:=TRUE;
		IF R_TRIG_Exeload.Q THEN
			NT_StartProcess_Load.START:=FALSE;
			NT_StartProcess_Load.PATHSTR:='C:\HZB\OpcIocShell\IDControlIOC\startTwinCATOPCServer.bat';
			Exe_load_step:=10;
		END_IF;
	10:
		IF LoadOpcIocTON.Q THEN
			NT_StartProcess_Load.START:=TRUE;
			Exe_load_step:=20;
		END_IF
	20:
		LoadOpcIocTON.IN:=FALSE;
		IF NT_StartProcess_Load.ERR THEN
			Exe_load_step:=0;
		ELSE
			Exe_load_step:=30;
		END_IF;
	30:
		IF NOT NT_StartProcess_Load.BUSY THEN
			NT_StartProcess_Load.START:=FALSE;
			Exe_Load_Done:=TRUE;
			Exe_load_step:=0;
		END_IF;
END_CASE;

NT_StartProcess_Load(
	NETID:='' ,
	PATHSTR:= ,
	DIRNAME:= , 
	COMNDLINE:= , 
	START:= ,
	ERRID=> );
END_ACTION

ACTION A_PosDiffDetectiion:
IF ABS(PosDiff_LeftTopLin_actual)>PosDiff_LeftTopLin THEN
	ErrorID:=201;
	Error:=TRUE;
	ErrorDescription:='ABS(PosDiff_LeftTopLin_actual)>PosDiff_LeftTopLin';
	FB_PlcEmergencyStop();
	LED_Error:=TRUE;
END_IF
IF ABS(PosDiff_RightTopLin_actual)>PosDiff_RightTopLin THEN
	ErrorID:=202;
	Error:=TRUE;
	ErrorDescription:='ABS(PosDiff_RightTopLin_actual)>PosDiff_RightTopLin';
	FB_PlcEmergencyStop();
	LED_Error:=TRUE;
END_IF
IF ABS(PosDiff_LeftBottomLin_actual)>PosDiff_LeftBottomLin THEN
	ErrorID:=203;
	Error:=TRUE;
	ErrorDescription:='ABS(PosDiff_LeftBottomLin_actual)>PosDiff_LeftBottomLin';
	FB_PlcEmergencyStop();
	LED_Error:=TRUE;
END_IF
IF ABS(PosDiff_RightBottomLin_actual)>PosDiff_RightBottomLin THEN
	ErrorID:=204;
	ErrorDescription:='ABS(PosDiff_RightBottomLin_actual)>PosDiff_RightBottomLin';
	Error:=TRUE;
	FB_PlcEmergencyStop();
	LED_Error:=TRUE;
END_IF
//
IF ABS(PosDiff_LeftTopLin_actual-PosDiff_RightTopLin_actual)>0.05 THEN
	ErrorID:=205;
	ErrorDescription:='ABS(PosDiff_LeftTopLin_actual-PosDiff_RightTopLin_actual)>0.05';
	Error:=TRUE;
	FB_PlcEmergencyStop();
	LED_Error:=TRUE;
ELSIF ABS(PosDiff_LeftBottomLin_actual-PosDiff_RightBottomLin_actual)>0.05 THEN
	ErrorID:=206;
	ErrorDescription:='ABS(PosDiff_LeftBottomLin_actual-PosDiff_RightBottomLin_actual)>0.05';
	Error:=TRUE;
	FB_PlcEmergencyStop();
	LED_Error:=TRUE;
END_IF
END_ACTION

ACTION A_RestartTC:
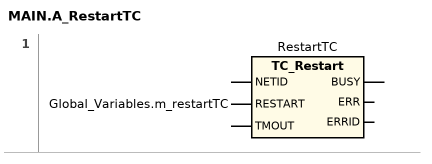
// NETWORK 1
RestartTC(RESTART := Global_Variables.m_restartTC); // TC_Restart
END_ACTION

ACTION A_SafePlcStartInit:
fb_ton0(PT:=t#1s);
fb_ton1(PT:=t#0.1s);
fb_ton2(PT:=t#0.1s);
fb_ton3(PT:=t#0.1s);

CASE SafeStatus OF
	0:
		IF COM_ERROR OR NOT Estop_Out THEN
			Err_Ack:=TRUE;
			fb_ton0.IN:=TRUE;
			SafeStatus:=1;
		ELSE
			SafePLCRunOK:=TRUE;
			SafeStatus:=0;
		END_IF
	1:
		IF fb_ton0.Q THEN
			Err_Ack:=FALSE;
			Safe_run:=TRUE;
			fb_ton1.IN:=TRUE;
			SafeStatus:=2;
		END_IF

	2:
		IF fb_ton1.Q THEN
			IF Estop_RunAndRestart=FALSE THEN
				Estop_RunAndRestart:=TRUE;
				fb_ton2.IN:=TRUE;
				SafeStatus:=3;
			END_IF
		END_IF
	3:
		IF fb_ton2.Q THEN
			IF Estop_RunAndRestart THEN
				Estop_RunAndRestart:=FALSE;
				fb_ton3.IN:=TRUE;
				SafeStatus:=4;
			END_IF
		END_IF
	4:
		IF fb_ton3.Q THEN
			IF Estop_Out THEN
				SafePLCRunOK:=TRUE;
				SafeStatus:=0;
			ELSE
				SafePLCRunOK:=FALSE;
				//Error:=TRUE;
				//ErrorId:=301;
				//ErrorDescription:='SafePLCRunOK fail';
			END_IF
		fb_ton0.IN:=FALSE;
		fb_ton1.IN:=FALSE;
		fb_ton2.IN:=FALSE;
		fb_ton3.IN:=FALSE;
		END_IF


END_CASE
END_ACTION

ACTION A_SetAxisPosition:
fb_ton4(PT:=t#0.5s);
CASE SetAxisPosState OF
	0:	(*FB_Set_AxisPosition*)
		FB_Set_AxisPosition(Execute:=TRUE);
		fb_ton4.IN:=TRUE;
		SetAxisPosState:=1;
	1:	(*wait*)
		FB_Set_AxisPosition();
		IF NOT FB_Set_AxisPosition.Done THEN		(*FB_Set_AxisPositionÃ»ÓÐÖ´ÐÐÍê£¬wait£¬³¬Ê±FB Error*)
			IF NOT fb_ton4.Q THEN
				SetAxisPosState:=1;
			ELSE
				SetAxisPosState:=99;
			END_IF
		ELSE
			SetAxisPosState:=88;
		END_IF
	88:
		SetAxisPosState:=0;
		SerAxisPositionDone:=TRUE;
		Error:=FALSE;
		ErrorID:=0;
		FB_Set_AxisPosition.Execute:=FALSE;
		fb_ton4.IN:=FALSE;
	99:
		SetAxisPosState:=99;
		SerAxisPositionDone:=FALSE;
		Error:=TRUE;
		FB_Set_AxisPosition.Execute:=FALSE;
		fb_ton4.IN:=FALSE;
		LED_Error:=TRUE;
		ErrorID:=401;
		ErrorDescription:='SetAxisPosition fail';
END_CASE
END_ACTION

ACTION A_SetLinearEncoderPositionBias:
//光栅positionBias补偿低温收缩量
IF CryogenicCompensationConditionsReady AND NOT CryogenicCompensationDone THEN
	PositionBias_LeftTop:=PositionBias_LeftTop+CryogenicCompensation_LeftTop;
	PositionBias_RightTop:=PositionBias_RightTop+CryogenicCompensation_RightTop;
	PositionBias_LeftBottom:=PositionBias_LeftBottom+CryogenicCompensation_LeftBottom;
	PositionBias_RightBottom:=PositionBias_RightBottom+CryogenicCompensation_RightBottom;
	CryogenicCompensationDone:=TRUE;
END_IF
//设置bias开始
A_SetLinearEncoderPositionBiasMC();
PositionBiasTON(PT:=T#0.1S);
CASE state_setLEPosBias OF
	0:
		PositionBiasTON.IN:=TRUE;
		IF MC_SetLEPosBias_LeftTop.Error OR MC_SetLEPosBias_RightTop.Error OR 
			MC_SetLEPosBias_LeftBottom.Error OR MC_SetLEPosBias_RightBottom.Error THEN
			state_setLEPosBias:=-100;
		ELSE 
			state_setLEPosBias:=1;
		END_IF
	1:
		IF NOT MC_SetLEPosBias_LeftTop.Done OR NOT MC_SetLEPosBias_RightTop.Done OR 
			NOT MC_SetLEPosBias_LeftBottom.Done OR NOT MC_SetLEPosBias_RightBottom.Done THEN
			MC_SetLEPosBias_LeftTop.Execute:=TRUE;
			MC_SetLEPosBias_RightTop.Execute:=TRUE;
			MC_SetLEPosBias_LeftBottom.Execute:=TRUE;
			MC_SetLEPosBias_RightBottom.Execute:=TRUE;
			state_setLEPosBias:=2;
		ELSE
			state_setLEPosBias:=-100;
		END_IF
	2:
		IF NOT MC_SetLEPosBias_LeftTop.Done OR NOT MC_SetLEPosBias_RightTop.Done OR 
			NOT MC_SetLEPosBias_LeftBottom.Done OR NOT MC_SetLEPosBias_RightBottom.Done THEN
			IF NOT PositionBiasTON.Q THEN
				state_setLEPosBias:=2;
			ELSE
				state_setLEPosBias:=-100;
			END_IF
		END_IF
		IF  MC_SetLEPosBias_LeftTop.Done AND MC_SetLEPosBias_RightTop.Done AND
			MC_SetLEPosBias_LeftBottom.Done AND MC_SetLEPosBias_RightBottom.Done THEN
			state_setLEPosBias:=88;
		END_IF	
		IF MC_SetLEPosBias_LeftTop.Error OR MC_SetLEPosBias_RightTop.Error OR 
			MC_SetLEPosBias_LeftBottom.Error OR MC_SetLEPosBias_RightBottom.Error THEN
			state_setLEPosBias:=-100;
		END_IF 
		
	88:
		PositionBiasTON.IN:=FALSE;
		PositionBiasDone:=TRUE;
	-100:
		PositionBiasTON.IN:=FALSE;
		PositionBiasDone:=FALSE;
		Error:=TRUE;
		ErrorId:=901;
		ErrorDescription:='Set LinearEncoderPositionBias Error';
		Plc_EmergencyStop:=FALSE;
END_CASE
END_ACTION

ACTION A_SetLinearEncoderPositionBiasMC:
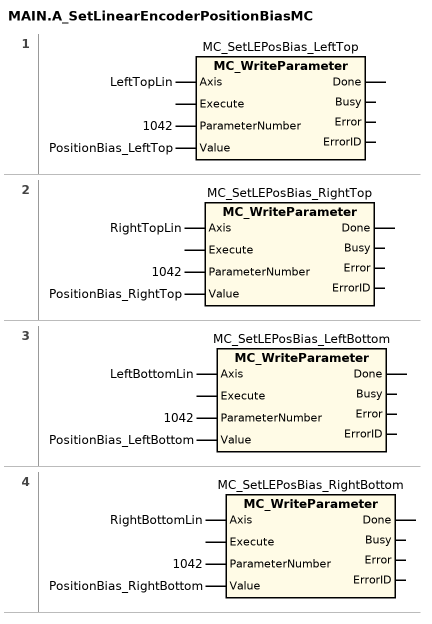
// NETWORK 1
MC_SetLEPosBias_LeftTop(Axis := LeftTopLin, ParameterNumber := 1042, Value := PositionBias_LeftTop); // MC_WriteParameter

// NETWORK 2
MC_SetLEPosBias_RightTop(Axis := RightTopLin, ParameterNumber := 1042, Value := PositionBias_RightTop); // MC_WriteParameter

// NETWORK 3
MC_SetLEPosBias_LeftBottom(Axis := LeftBottomLin, ParameterNumber := 1042, Value := PositionBias_LeftBottom); // MC_WriteParameter

// NETWORK 4
MC_SetLEPosBias_RightBottom(
    Axis := RightBottomLin,
    ParameterNumber := 1042,
    Value := PositionBias_RightBottom); // MC_WriteParameter
END_ACTION

END_PROGRAM

(* stored: Version 1.1.0.1, ProductVersion 3.1.4024.6
   POU MAIN: Id {9221b602-3f7e-4757-b581-54b56182ad8f}, SpecialFunc None
   Folder Axis: Id {1f5db9b2-f074-43bd-a7a5-f28b002c6ac6}
   Folder Check: Id {79c48f21-8e44-4159-8773-87594d6e7620}
   Folder Driver: Id {06d9eaf4-b0e1-444b-9d9d-89e6e18ffc32}
   Folder LinearEncoder: Id {4f24c8b2-fa71-4a79-b365-8e83326d2610}
   Folder Recipe: Id {c556f121-0220-445e-afd2-6e585e1080be}
   Folder Safe: Id {8d52a6a5-8a59-474d-a357-67246f4286de}
   Folder TC: Id {4ef3e57e-ed4b-4379-8b8b-cf198d1ecdc5}
   Folder Temperature: Id {ca29eaee-6597-4656-befc-70156b197af2}
   Action A_CheckHardwareEmergencyStopStatus: Id {c59a955b-0a8f-43a7-a0e7-3ab11b3d5ab6}
   Action A_CheckKillSwitch: Id {158eed83-fba1-4051-b569-3585448d2a5a}
   Action A_CheckLimitSwitch: Id {1026ae85-58e3-4004-8dd3-becfab0085f9}
   Action A_CryogenicCompensationMonitoring: Id {196f46d5-b4be-43fe-a564-735eda66c49f}
   Action A_GetDriverStatus: Id {e05cf975-7b3e-4430-bb2e-a308f4391f1b}
   Action A_GetDriverStatusMC: Id {2d8972a4-2924-4445-a68a-757b585b0760}
   Action A_GetTemperatureSensorsData: Id {d73fb87c-9e06-4b36-8cf6-68d5032eab30}
   Action A_InitAxisParameters: Id {a92c2dd6-12b0-4a71-a4bc-d7afbc965cb4}
   Action A_InitRecipeParameters: Id {6aa76980-7ae7-46e7-9688-f94b6fa6510d}
   Action A_KillOpcIocShellExe: Id {e0252576-ad9e-49ed-bcc5-7f64aacd5ffe}
   Action A_LoadOpcIocShellExe: Id {e69e9ea4-205f-45b3-85e7-e1c1b3150dfb}
   Action A_PosDiffDetectiion: Id {e857c546-d367-4f19-9434-ed29c144eb6f}
   Action A_RestartTC: Id {737d9420-c364-46ec-805e-ce283c214994}
   Action A_SafePlcStartInit: Id {4d1a8480-9923-4117-8ca7-ea613a82dfad}
   Action A_SetAxisPosition: Id {eb32aedd-8f01-44b1-96a9-73f233ea8548}
   Action A_SetLinearEncoderPositionBias: Id {6f3d3f8e-255d-4e09-853f-5fdf91122229}
   Action A_SetLinearEncoderPositionBiasMC: Id {d950edd3-252b-4c3c-9e26-a84e2707fa62} *)
